(* LS Electric XG5000 project: 241011_실습PLC와연동해서램프켜기WITH타이머 *)
(* PLC LSPLC *)

PROGRAM NewProgram (* task: 스캔 프로그램 *)
VAR
    MX AT %MW0 : INT;
    NUM : STRING;
    S1 : STRING;
    S2 : STRING;
    STR : STRING;
    T1 : TON;
    TIME1 : TIME;
END_VAR

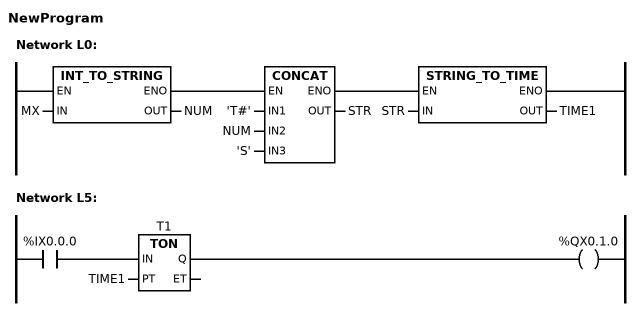
(* Rung L0 *)
NUM := INT_TO_STRING(MX);
STR := CONCAT('T#', NUM, 'S');
TIME1 := STRING_TO_TIME(STR);
(* Rung L5 *)
T1(IN := %IX0.0.0, PT := TIME1);
%QX0.1.0 := T1.Q;
END_PROGRAM